FUNCTION_BLOCK DataTypesFloatingPoints (* Template for an empty basic function block *)
  (* Standard: 61499-2; Description: Normal just propagates the input to the output Internal: sets the output from inside to pi and e Copyright (c) 2019 Jan Holzweber This program and the accompanying materials are made available under the terms of the Eclipse Public License 2.0 which is available at https://www.eclipse.org/legal/epl-2.0/ SPDX-License-Identifier: EPL-2.0 *)
  (* Version 1.0, 2019-06-05, jholz *)
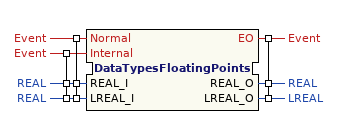
  EVENT_INPUT
    Normal WITH REAL_I, LREAL_I;
    Internal WITH REAL_I, LREAL_I;
  END_EVENT
  EVENT_OUTPUT
    EO WITH REAL_O, LREAL_O;
  END_EVENT
  VAR_INPUT
    REAL_I : REAL;
    LREAL_I : REAL;
  END_VAR
  VAR_OUTPUT
    REAL_O : REAL;
    LREAL_O : LREAL;
  END_VAR
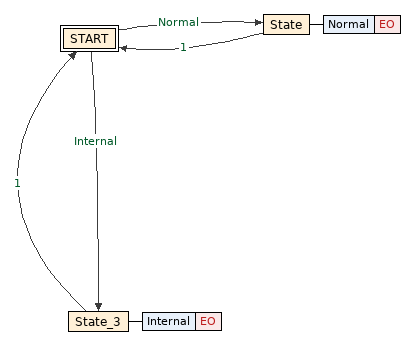
  EC_STATES
    START; (* Initial State *)
    State : Normal -> EO;
    State_3 : Internal -> EO;
  END_STATES
  EC_TRANSITIONS
    START TO State := Normal;
    State TO START := 1;
    START TO State_3 := Internal;
    State_3 TO START := 1;
  END_TRANSITIONS
  ALGORITHM Normal IN ST: (* new algorithm *)
REAL_O:=REAL_I;
LREAL_O :=LREAL_I;
  END_ALGORITHM
  ALGORITHM Internal IN ST: (* new algorithm *)
REAL_O:=3.14159265359;
LREAL_O :=2.7182818;
  END_ALGORITHM
END_FUNCTION_BLOCK
